FUNCTION_BLOCK FB_KPI_CaseEfficiency
VAR_INPUT
	bUpdateItemData		: 	BOOL;
	bItemSuccessful		:	 BOOL;
END_VAR
VAR_IN_OUT
	stItemInspection		: 	ST_KPI_InspectionEfficency;
END_VAR
VAR_OUTPUT
END_VAR
VAR
	rtrigUpdateItemData	:	 R_TRIG;
END_VAR

rtrigUpdateItemData(CLK:= bUpdateItemData);

IF rtrigUpdateItemData.Q THEN

	stItemInspection.ProcessedTotal :=  stItemInspection.ProcessedTotal + 1;
		IF bItemSuccessful THEN
			stItemInspection.ProcessedSuccessful := stItemInspection.ProcessedSuccessful + 1;
		ELSE
			stItemInspection.ProcessedRejected := stItemInspection.ProcessedRejected + 1;
		END_IF
END_IF

stItemInspection.ProcessedEfficiency := F_SafeDIV(stItemInspection.ProcessedSuccessful  * 100,  stItemInspection.ProcessedTotal);
stItemInspection.ProcessedEfficiency :=LIMIT(0, stItemInspection.ProcessedEfficiency, 100);

END_FUNCTION_BLOCK

(* stored: Version 1.1.0.1, ProductVersion 3.1.4024.15
   POU FB_KPI_CaseEfficiency: Id {9375ae1b-7a02-4976-909e-db08e779eaef}, SpecialFunc None *)
